{attribute addProperty ShortName "CU00x"}
{attribute addProperty Name "Controlled unit template"}
FUNCTION_BLOCK CU00x EXTENDS CUBase
VAR
    _cuData      : REFERENCE TO CU00xProcessData;
    _processData : ProcessDataManager(THIS^);
    _components  : CU00xComponents := (Parent := THIS^);
	{attribute addProperty Name "<#AUTOMAT#>"}
	{attribute addProperty ToolTip "<#Starts automatic sequence. Before start you need to perform grounding sequence.#>"}
    _automat     : CU00xAutomat(THIS^, TcoCore.eRestoreMode.None);	
	{attribute addProperty Name "<#GROUND#>"}
	{attribute addProperty ToolTip "<#Brings the device into basic position.#>"}
    _ground      : CU00xGround(THIS^, TcoCore.eRestoreMode.None);
	{attribute addProperty Name "<#MANUAL#>"}
	{attribute addProperty ToolTip "<#Start manual/Service mode#>"}
    _manual      : CU00xManual(THIS^);
END_VAR

_processData();

_automat.Task.Enabled := _ground.GroundDone;
_automat();

_ground.Task.Enabled := NOT _ground.Task.Done;
_ground();

_manual.Task.Enabled := TRUE;
_manual();

UpdateInfo();

PROPERTY Automat : REFERENCE TO TcoTaskedSequencer
GET
Automat REF= _automat;
END_GET
END_PROPERTY

METHOD CancelGround
VAR_INPUT
END_VAR
_ground.CancelGround();
END_METHOD

PROPERTY Components : REFERENCE TO CU00xComponents
GET
Components REF= _components;
END_GET
END_PROPERTY

PROPERTY Ground : REFERENCE TO TcoTaskedSequencer
GET
Ground REF= _ground;
END_GET
END_PROPERTY

METHOD InitializeComponents : BOOL
END_METHOD

PROPERTY Manual : REFERENCE TO TcoTaskedService
GET
Manual REF= _manual;
END_GET
END_PROPERTY

PROPERTY ProcessDataManager : REFERENCE TO ProcessDataManager
GET
ProcessDataManager REF= _processData;
END_GET
END_PROPERTY

PROPERTY Technology : REFERENCE TO Technology
GET
VAR
    _technology : POINTER TO Technology;
END_VAR
IF __QUERYPOINTER(Parent, _technology) THEN // Check if _Parent is Station001
    Technology REF= _technology^;              // If the check is successful dereference a pointer. simlar to THIS^ or SUPER^
END_IF
END_GET
END_PROPERTY

END_FUNCTION_BLOCK

(* stored: Version 1.1.0.1, ProductVersion 3.1.4024.9
   POU CU00x: Id {c8fb8f62-fa26-41d3-a5d2-3cc70d4e8555}, SpecialFunc None
   Property Automat: Id {395ce4fa-38ae-46a5-9c91-86a9f1bcbbc2}
   Get Get: Id {ca2cc00e-064b-48f3-a4fa-26832ebfc11a}
   Method CancelGround: Id {2a6a329c-2fd1-4101-9cbb-b4d390744e07}
   Property Components: Id {7133061c-46ce-4913-b91f-5deb41132b8c}
   Get Get: Id {d34691d4-caf0-4f1c-9ccf-b26a123c3f8f}
   Property Ground: Id {49f8c54b-7096-4ee9-be7f-1b5b62c4c097}
   Get Get: Id {8480f5d4-4535-49b0-b4be-60aa7bf89b76}
   Method InitializeComponents: Id {5a5fba3f-8ac9-4756-a6a5-163b8c66ad67}
   Property Manual: Id {3362f8a1-5828-47e8-a58f-b7a215df59dc}
   Get Get: Id {e78cfa35-d5c6-462d-8720-3fee9ea9f425}
   Property ProcessDataManager: Id {9c871fab-0088-44ca-b24f-778dec392de1}
   Get Get: Id {95b32202-bc09-4e9e-9cf9-08fc5dcf9bf8}
   Property Technology: Id {0e688a71-683a-45e9-ad1b-4b5b04f7d71e}
   Get Get: Id {6127ba68-461c-4b3d-aa46-b1cbb1962cc4} *)
